// TIA Portal V17 export
// export: Created 2025-01-20T10:26:49.4056979Z, ExportSetting WithDefaults, DisplayName Totally Integrated Automation Portal, DisplayVersion V17 Update 7, DisplayName TIA Portal Openness, DisplayVersion V17 Update 7, DisplayName TIA Portal Version Control Interface, DisplayVersion V17, DisplayName SINAMICS Startdrive Advanced, DisplayVersion V17 SP2, DisplayName SINAMICS Startdrive G110M, G120, G120C, G120D, G120P, G115D, DisplayVersion V17 SP2, DisplayName SINAMICS Startdrive G130, G150, S120, S150, SINAMICS MV, S210, DisplayVersion V17 SP2, DisplayName STEP 7 Professional, DisplayVersion V17 Update 7, DisplayName STEP 7 Safety, DisplayVersion V17 Update 6, DisplayName WinCC Professional, DisplayVersion V17 Update 7
VAR_GLOBAL   // PLC tag table "Default tag table"
   Tag_1 AT %M1.0 : Bool;
   Tag_2 AT %M2.0 : Bool;
   Tag_3 AT %M3.0 : Bool;
   Tag_4 AT %M10.0 : Bool;
   Tag_5 AT %M20.0 : Bool;
   Tag_6 AT %M1.1 : Bool;
   Tag_7 AT %M23.0 : Bool;
END_VAR
